{attribute 'linkalways'} 
{attribute 'no_explicit_call' := 'This FB is a CLASS and must be accessed using methods or properties'}
{attribute 'enable_dynamic_creation'}
FUNCTION_BLOCK MockStructuredDatatype_TIMESTRUCT EXTENDS StructuredDatatypeBase
VAR
	localData : TIMESTRUCT;
	activeData : REFERENCE TO TIMESTRUCT REF= localData;
	_wYear : _WORD(localData.wYear);
	_wMonth : _WORD(localData.wMonth);
	_wDayOfWeek : _WORD(localData.wDayOfWeek);
	_wDay : _WORD(localData.wDay);
	_wHour : _WORD(localData.wHour);
	_wMinute : _WORD(localData.wMinute);
	_wSecond : _WORD(localData.wSecond);
	_wMilliseconds : _WORD(localData.wMilliseconds);
END_VAR

PROPERTY PUBLIC Address : PVOID
GET
Address := ADR(activeData);
END_GET
END_PROPERTY

METHOD PUBLIC ClearReference
VAR_INPUT
END_VAR
activeData REF= localData;
SetMemberReference();
END_METHOD

METHOD PUBLIC Clone : I_Datatype
VAR
    pClone : POINTER TO MockStructuredDatatype_TIMESTRUCT;
END_VAR
pClone := __NEW(MockStructuredDatatype_TIMESTRUCT());
pClone^.Value := Value;
Clone := pClone^;
END_METHOD

METHOD FB_init : BOOL
VAR_INPUT
	bInitRetains : BOOL; // if TRUE, the retain variables are initialized (warm start / cold start)
	bInCopyCode : BOOL;  // if TRUE, the instance afterwards gets moved into the copy code (online change)
END_VAR
SetMemberReference();
AddMember('wYear',_wYear);
AddMember('wMonth',_wMonth);
AddMember('wDayOfWeek',_wDayOfWeek);
AddMember('wDay',_wDay);
AddMember('wHour',_wHour);
AddMember('wMinute',_wMinute);
AddMember('wSecond',_wSecond);
AddMember('wMilliseconds',_wMilliseconds);
END_METHOD

PROPERTY PUBLIC Identifier : T_MAXSTRING
GET
Identifier := 'TIMESTRUCT';
END_GET
END_PROPERTY

METHOD PUBLIC MakeReferenceTo
VAR_INPUT
	ReferenceTarget : REFERENCE TO TIMESTRUCT;
END_VAR
activeData REF= ReferenceTarget;
SetMemberReference();
END_METHOD

METHOD PROTECTED SetMemberReference
VAR_INPUT
END_VAR
_wYear.MakeReferenceTo(activeData.wYear);
_wMonth.MakeReferenceTo(activeData.wMonth);
_wDayOfWeek.MakeReferenceTo(activeData.wDayOfWeek);
_wDay.MakeReferenceTo(activeData.wDay);
_wHour.MakeReferenceTo(activeData.wHour);
_wMinute.MakeReferenceTo(activeData.wMinute);
_wSecond.MakeReferenceTo(activeData.wSecond);
_wMilliseconds.MakeReferenceTo(activeData.wMilliseconds);
END_METHOD

PROPERTY PUBLIC Size : UDINT
GET
Size := SIZEOF(activeData);
END_GET
END_PROPERTY

METHOD TryMakeReferenceTo : BOOL
VAR_INPUT
	Target : I_Datatype;
END_VAR
VAR
	pTargetData : POINTER TO TIMESTRUCT;
END_VAR
IF NOT IsEquivalentTo(Target) THEN
	RETURN;
END_IF

pTargetData := Target.Address;
activeData REF= pTargetData^;
SetMemberReference();
TryMakeReferenceTo := TRUE;
END_METHOD

PROPERTY PUBLIC Value : REFERENCE TO TIMESTRUCT
GET
Value REF= activeData;
END_GET
END_PROPERTY

PROPERTY PUBLIC wDay : Reference to _WORD
GET
wDay REF= _wDay;
END_GET
END_PROPERTY

PROPERTY PUBLIC wDayOfWeek : Reference to _WORD
GET
wDayOfWeek REF= _wDayOfWeek;
END_GET
END_PROPERTY

PROPERTY PUBLIC wHour : Reference to _WORD
GET
wHour REF= _wHour;
END_GET
END_PROPERTY

PROPERTY PUBLIC wMilliseconds : Reference to _WORD
GET
wMilliseconds REF= _wMilliseconds;
END_GET
END_PROPERTY

PROPERTY PUBLIC wMinute : Reference to _WORD
GET
wMinute REF= _wMinute;
END_GET
END_PROPERTY

PROPERTY PUBLIC wMonth : Reference to _WORD
GET
wMonth REF= _wMonth;
END_GET
END_PROPERTY

PROPERTY PUBLIC wSecond : Reference to _WORD
GET
wSecond REF= _wSecond;
END_GET
END_PROPERTY

PROPERTY PUBLIC wYear : Reference to _WORD
GET
wYear REF= _wYear;
END_GET
END_PROPERTY

END_FUNCTION_BLOCK

(* stored: Version 1.1.0.1, ProductVersion 3.1.4024.13
   POU MockStructuredDatatype_TIMESTRUCT: Id {00a68b55-ff51-46df-9d73-ac621162111d}, SpecialFunc None
   Folder Constructor: Id {42abd6e4-a633-4990-9b21-a90233d3a0f1}
   Folder Protected: Id {5cb501b4-a7fc-4879-861f-237dc8aca9f6}
   Property Address: Id {5efd1043-d12a-4a1c-96a6-3e3d077a4e76}
   Get Get: Id {89e6f9ed-0d4f-4ef8-8f90-aa6cd4cf603f}
   Method ClearReference: Id {c9759825-bc7f-4d17-b88c-e8f9ba8b3096}
   Method Clone: Id {d0d9a843-6b3a-49f6-8499-e5c35e3212d4}
   Method FB_init: Id {3be0afc5-fae0-48d2-9d94-65681c9f8c90}
   Property Identifier: Id {d7c884d8-6e24-450e-80b7-209269372358}
   Get Get: Id {c7304741-a6df-49d0-bf8e-cec94160f0d2}
   Method MakeReferenceTo: Id {c4ea6cc4-d46d-49d0-8373-ec987167bfca}
   Method SetMemberReference: Id {f0fbce4d-a970-498b-8341-ee07a8dd1576}
   Property Size: Id {c4efa261-7e9e-45af-a7d5-66b610c59260}
   Get Get: Id {b1db2f6d-15a2-433c-9491-d79099775a11}
   Method TryMakeReferenceTo: Id {a6a884e8-bc8f-43a4-b9d3-3bad96a93c94}
   Property Value: Id {4f218980-58c3-4e2f-81d7-18189a9547e2}
   Get Get: Id {bc9f5041-5b22-4cbf-8ef0-457308879e06}
   Property wDay: Id {5839d803-55c0-4b59-8e7c-8f28bf44ae20}
   Get Get: Id {ca35cd4a-1f2f-4670-b368-300df08006d7}
   Property wDayOfWeek: Id {5663dd0e-b036-431a-a13f-c4ee35f8a962}
   Get Get: Id {1c819719-b504-43dd-9e49-dff285f355b5}
   Property wHour: Id {74926152-3d10-4e22-a338-019763fb1dfc}
   Get Get: Id {e3b6db93-12ed-4aaf-a96d-edf5cb3b01c4}
   Property wMilliseconds: Id {7e371212-62b8-43a8-846e-d67d05a6cb04}
   Get Get: Id {4b9ab695-0aa9-47c6-885c-b6b33453bb6e}
   Property wMinute: Id {0b10f29f-9b2b-472c-b5cc-26d4dc83cf2e}
   Get Get: Id {abb79c73-c4ac-4398-b90c-bc981a85d1fb}
   Property wMonth: Id {3caac212-f448-4337-a442-a39670cfae85}
   Get Get: Id {08cf691c-a5b8-446e-bfb2-4d2588958291}
   Property wSecond: Id {058e1083-9bc0-4522-ab9a-a2c0264ece67}
   Get Get: Id {8357e256-ee61-48ad-8962-7e8fe2211e9d}
   Property wYear: Id {e241ab71-65fb-4bbf-982b-58c16d3e7e10}
   Get Get: Id {f7b878c2-bfc2-43b2-a2a8-660f819b5677} *)
